FUNCTION_BLOCK RunGradeOutput EXTENDS RunUnitSlave
VAR
	axisMoving : POINTER TO RunAxis;
	holder : POINTER TO RunCylinder;
	axisVertical : POINTER TO RunCylinder;
	clamper : POINTER TO RunCylinder;	
	//
	ptCommandReady : POINTER TO ParameterSet;
	ptCommandOK : POINTER TO ParameterSet;
	ptCommandNG : POINTER TO ParameterSet;
	//
	block : MaterialBlock;
	ptDesitination : POINTER TO parameterset;
END_VAR
VAR PERSISTENT
	isQuery : bool ; //whether query material data when material income
END_VAR

//Ng/OK output mechanism
SUPER^();

CASE outputState OF 
	//-------------------------Initialize
	eSpecialStates.INITIAL_BEGIN:
		transitionByte.0 := holder^.Execute(eCylinderCommands.COMMAND_A);
		transitionByte.1 := clamper^.Execute(eCylinderCommands.COMMAND_A);
		bSerialTransition := (transitionByte = 16#3);
	eSpecialStates.INITIAL_STATE_1:
		bSerialTransition :=  axisVertical^.Execute(eCylinderCommands.COMMAND_A);
	eSpecialStates.INITIAL_STATE_2:
		IF axisMoving^.ExecuteParameter(ptCommandReady) THEN
			NextState := eSpecialStates.INITIAL_END;
		END_IF
	//------------------------Working
	eSpecialStates.SLAVE_ENTER_PROCEDURE:
		//---------------
		//	Material infor exchanging
		//---------------
		SlotLast^.Id := SlotBase^.Id; //the clamper work station
		SlotLast^.Valid := SlotLast^.Valid;
		IF SlotLast^.Valid THEN
			SlotLast^.Act := isQuery; //query grade
			bSerialTransition := TRUE;
		ELSE
			NextState := eSpecialStates.SLAVE_WORK_DONE;		
		END_IF
	16#201:
		bSerialTransition:=axisVertical^.Execute(eCylinderCommands.COMMAND_B); //down
	16#202:
		bSerialTransition:=holder^.Execute(eCylinderCommands.COMMAND_B); //hold
	16#203:
		bSerialTransition:=clamper^.Execute(eCylinderCommands.COMMAND_B); //clamper relase
	16#204:
		bSerialTransition:=axisVertical^.Execute(eCylinderCommands.COMMAND_A); //up
	16#205:
		bSerialTransition:=clamper^.Execute(eCylinderCommands.COMMAND_A); //clamper return
		IF bSerialTransition THEN
			workingSignal^ := FALSE; //release conveyor
		END_IF
	16#206:
		bSerialTransition := NOT SlotLast^.Act; //wait until query over
		IF bSerialTransition THEN
			block := SlotLast^.Data;
			CASE block.data[0] OF
				0:
					//ng
					ptDesitination := ptCommandNG;
				1:
					//ok
					ptDesitination := ptCommandOK;
			END_CASE
		END_IF
	16#207:
		IF axisMoving^.ExecuteParameter(ptDesitination) THEN
			//according TO grade TO MOVE
			NextState := 16#210;
		END_IF
	//-------------------Drop
	16#210: 
		bSerialTransition:=holder^.Execute(eCylinderCommands.COMMAND_A); //release
	16#211:
		IF axisMoving^.ExecuteParameter(ptCommandReady) THEN
			NextState := 0;
		END_IF
END_CASE

METHOD FB_init : BOOL
VAR_INPUT
	bInitRetains : BOOL; // if TRUE, the retain variables are initialized (warm start / cold start)
	bInCopyCode : BOOL;  // if TRUE, the instance afterwards gets moved into the copy code (online change)
	
	argParent : POINTER TO RunUnitGeneric;
	argSlotBase : POINTER TO RunMaterial;
	argSlotLast : POINTER TO RunMaterial;
	
	argWorkingSignal : POINTER TO BOOL;
	
	argAxisMoving : POINTER TO RunAxis;
	
	argHolder : POINTER TO RunCylinder;
	argAxisVertical : POINTER TO RunCylinder;
	argClamper : POINTER TO RunCylinder;
	
END_VAR
VAR CONSTANT
	indexReady : INT := 1;
	indexOK : INT := 2;
	indexNG : INT := 3;
END_VAR
//initialize 
Parent := argParent;
SlotBase := argSlotBase;
SlotLast := argSlotLast;
//
IF bInitRetains THEN
	NextState := eSpecialStates.INITIAL_BEGIN;
END_IF

workingSignal := argWorkingSignal; //link

//Axis
axisMoving := argAxisMoving;
ptCommandReady := ADR(axisMoving^.ptpCommands[indexReady]);
ptCommandOK := ADR(axisMoving^.ptpCommands[indexOK]);
ptCommandNG := ADR(axisMoving^.ptpCommands[indexNG]);

holder := argHolder;
axisVertical := argAxisVertical;
clamper := argClamper;
END_METHOD

END_FUNCTION_BLOCK

(* stored: Version 1.1.0.1, ProductVersion 3.1.4022.10
   POU RunGradeOutput: Id {3be266a6-2ed3-4d2f-a14a-5486dca5768b}, SpecialFunc None
   Method FB_init: Id {16d063af-8ad4-4db2-a192-b68a7dec8537} *)
